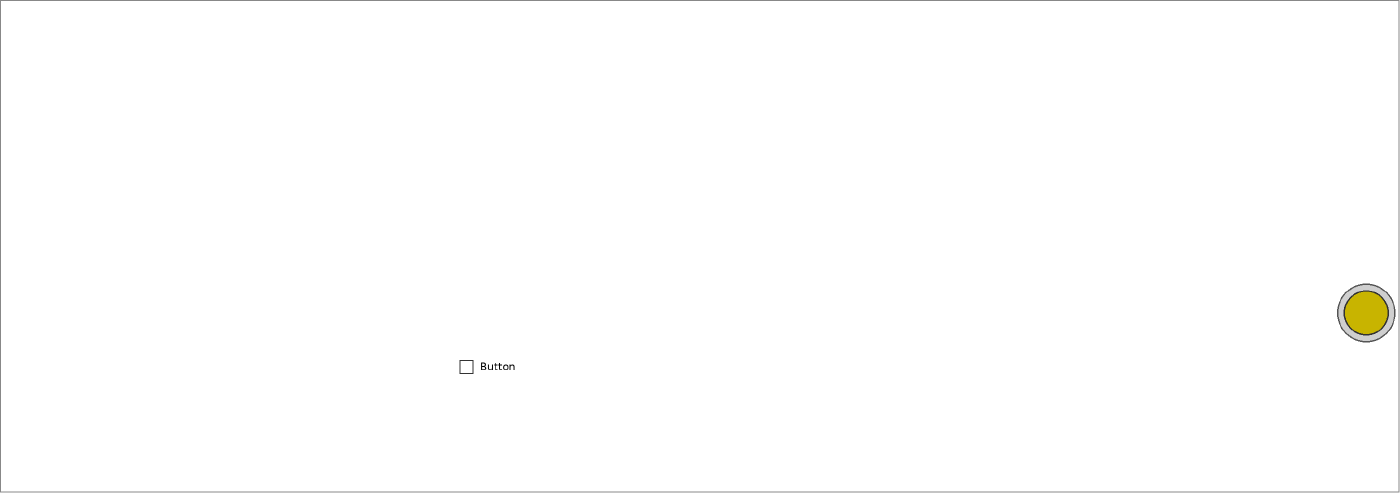
VISUALIZATION Visualization  // 1453x512
    Checkbox (475,250 326x262), "Button", variable: MAIN.bButton
    Lamp1 (1383,290 70x70), variable: MAIN.bLED, style: Lamp-Lamp1-Yellow
END_VISUALIZATION

(* stored: Version 1.1.0.1
   Visu Visualization: Id {759a59d8-e12f-49a7-85a3-37ca417e3789} *)
